// TIA Portal project "cyclic interrupt ile flasor" (V16)

(* hardware
DEVICE "S7-1200 station_1"  S7-1200 Station
   slot 0: "Rack_0"  S7-1200 Rack  Rack  V1.0
   slot 1: "PLC_1"  CPU 1217C DC/DC/DC  6ES7 217-1AG40-0XB0  V4.4
*)

// ===== PLC "PLC_1"  CPU 1217C DC/DC/DC =====

VAR_GLOBAL   // PLC tag table "Default tag table"
   "System_Byte" AT %MB1 : Byte;
   "FirstScan" AT %M1.0 : Bool;
   "DiagStatusUpdate" AT %M1.1 : Bool;
   "AlwaysTRUE" AT %M1.2 : Bool;
   "AlwaysFALSE" AT %M1.3 : Bool;
   "Clock_Byte" AT %MB0 : Byte;
   "Clock_10Hz" AT %M0.0 : Bool;
   "Clock_5Hz" AT %M0.1 : Bool;
   "Clock_2.5Hz" AT %M0.2 : Bool;
   "Clock_2Hz" AT %M0.3 : Bool;
   "Clock_1.25Hz" AT %M0.4 : Bool;
   "Clock_1Hz" AT %M0.5 : Bool;
   "Clock_0.625Hz" AT %M0.6 : Bool;
   "Clock_0.5Hz" AT %M0.7 : Bool;
   "trg_1" AT %M2.0 : Bool;
   "bi_saniye" AT %M2.1 : Bool;
   "Tag_1" AT %Q0.0 : Bool;
   "dume_1" AT %M2.2 : Bool;
   "den" AT %MW4 : Int;
   "taata" AT %M2.3 : Bool;
   "ktp" AT %M2.4 : Bool;
   "buton" AT %M2.5 : Bool;
   "trg_2" AT %M2.6 : Bool;
   "aa" AT %M2.7 : Bool;
END_VAR

ORGANIZATION_BLOCK "Main"   // OB1, LAD, ProgramCycle
TITLE = "Main Program Sweep (Cycle)"
{ S7_Optimized_Access := 'TRUE' }
VERSION : 0.1
   VAR_INPUT
      Initial_Call : Bool;   // Initial call of this OB
      Remanence : Bool;   // =True, if remanent data are available
   END_VAR
BEGIN
END_ORGANIZATION_BLOCK

ORGANIZATION_BLOCK "Cyclic interrupt"   // OB30, LAD, CyclicInterrupt
{ S7_Optimized_Access := 'TRUE' }
VERSION : 0.1
// cycle her çalıştığında sadece bir tarama yapar. Yani başa yükselen kenar koymaya gerek yok.
   VAR_INPUT
      Initial_Call : Bool;   // Initial call of this OB
      Event_Count : Int;   // Events discarded
   END_VAR
   VAR_TEMP   // added for the SCL form of the ladder/FBD networks
      _w1 : Bool;
   END_VAR
BEGIN

REGION Network 1
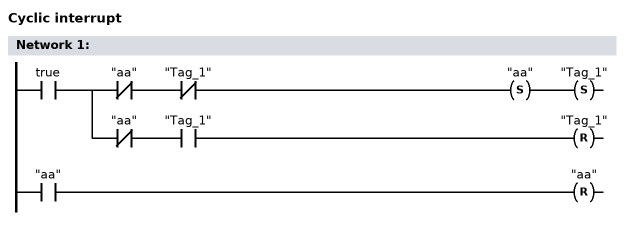
   RUNG wire#powerrail
      Contact( true )
      wire#w1
      I_Contact( "aa" )
      I_Contact( "Tag_1" )
      S_Coil( "aa" )
      S_Coil( "Tag_1" )
   END_RUNG
   RUNG wire#w1
      I_Contact( "aa" )
      Contact( "Tag_1" )
      R_Coil( "Tag_1" )
   END_RUNG
   RUNG wire#powerrail
      Contact( "aa" )
      R_Coil( "aa" )
   END_RUNG
   // the same network as SCL:
   #_w1 := true AND NOT "aa" AND NOT "Tag_1";
   IF #_w1 THEN
       "aa" := TRUE;
       "Tag_1" := TRUE;
   END_IF;
   IF true AND NOT "aa" AND "Tag_1" THEN "Tag_1" := FALSE; END_IF;
   IF "aa" THEN "aa" := FALSE; END_IF;
END_REGION
END_ORGANIZATION_BLOCK